FUNCTION AxesDeltaUnitsToDeg : LREAL
VAR_INPUT
    units : AxesDeltaUnits;
    value : LREAL;
END_VAR
VAR
END_VAR

CASE units OF
    AxesDeltaUnits.RADIANS:
        AxesDeltaUnitsToDeg := RAD_TO_DEG(value);
    AxesDeltaUnits.DEGREES:
        AxesDeltaUnitsToDeg := value;  
END_CASE

END_FUNCTION

(* stored: Version 1.1.0.1, ProductVersion 3.1.4019.2
   POU AxesDeltaUnitsToDeg: Id {0d906718-a020-49c6-b676-63ec91b9c37c}, SpecialFunc None *)
